  MoveL 646 to (-11.76, 196.67, 20) mm, rotated rx 135.83 ry -73.06 rz -38.46 deg; joints [-4.295, 33.165, -46.242, 103.942, -105.646, 46.988, -1571.54]
  MoveL 647 to (-16.38, 197.8, 10) mm, rotated rx 132.74 ry -74.34 rz -42.53 deg; joints [-4.695, 34.359, -48.607, 102.356, -105.543, 42.262, -1567.469]
  MoveL 648 to (-20.49, 199.16, 0) mm, rotated rx 132.74 ry -74.34 rz -42.53 deg; joints [-5.02, 34.493, -48.595, 102.456, -105.203, 42.34, -1567.469]
  Set speed (1000.0 mm/s)
  MoveL 649 to (-20.49, 199.16, 0) mm, rotated rx 132.74 ry -74.34 rz -42.53 deg; joints [-5.02, 34.493, -48.595, 102.456, -105.203, 42.34, -1567.469]
  Set speed (1000.0 mm/s)
